FUNCTION_BLOCK MTR_CNTRL_POS (* Basic Function Block Type *)
  (* Standard: 61499-2 *)
  (* Version 0.3, 2009-09-15, JHC, Holobloc Inc, Changed transition priorities. *)
  (* Version 0.2, 2003-12-04, JHC, Rockwell Automation, Renamed for better indexing. *)
  (* Version 0.1, 2002-11-05, JHC, Rockwell Automation, Corrected missing ST element in Algorithm REQ. *)
  (* Version 0.0, 2000-05-30, JHC, Rockwell Automation *)
  (* Compiler header: package fb.rt.template; *)
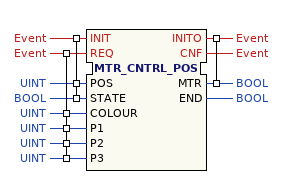
  EVENT_INPUT
    INIT WITH POS, STATE; (* Initialization Request *)
    REQ WITH COLOUR, P1, P2, P3;
  END_EVENT
  EVENT_OUTPUT
    INITO WITH MTR; (* Initialization Confirm *)
    CNF;
  END_EVENT
  VAR_INPUT
    POS : UINT;
    STATE : BOOL;
    COLOUR : UINT;
    P1 : UINT;
    P2 : UINT;
    P3 : UINT;
  END_VAR
  VAR_OUTPUT
    MTR : BOOL; (* Output event qualifier *)
    END : BOOL;
  END_VAR
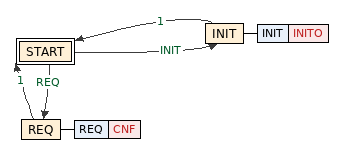
  EC_STATES
    START; (* Initial State *)
    INIT : INIT -> INITO; (* Initialization *)
    REQ : REQ -> CNF;
  END_STATES
  EC_TRANSITIONS
    INIT TO START := 1;
    START TO INIT := INIT;
    START TO REQ := REQ;
    REQ TO START := 1;
  END_TRANSITIONS
  ALGORITHM INIT IN ST: (* Initialization algorithm *)
MTR:=FALSE;
END:=FALSE;
  END_ALGORITHM
  ALGORITHM REQ IN ST:
IF STATE THEN
  MTR:=TRUE;
	IF COLOUR=1 THEN
		IF POS<P1 THEN
			MTR:=TRUE;
		ELSE
			MTR:=FALSE;
			END:=TRUE;
		END_IF;
	END_IF;
	IF COLOUR=2 THEN
		IF POS<P2 THEN
			MTR:=TRUE;
		ELSE
			MTR:=FALSE;
			END:=TRUE;
		END_IF;
	END_IF;
	IF COLOUR=3 THEN
		IF POS<P3 THEN
			MTR:=TRUE;
		ELSE
			MTR:=FALSE;
			END:=TRUE;
		END_IF;
	END_IF;
END_IF;
  END_ALGORITHM
END_FUNCTION_BLOCK
